FUNCTION_BLOCK CU010ExampleCompositComponent EXTENDS TcoCore.TcoComponent
VAR_INPUT
END_VAR
VAR_OUTPUT
END_VAR
VAR
END_VAR

END_FUNCTION_BLOCK

(* stored: Version 1.1.0.1
   POU CU010ExampleCompositComponent: Id {0ed64ab4-648a-43c3-886f-aaf92674c0f7}, SpecialFunc None *)
